FUNCTION_BLOCK FB_Dictionary IMPLEMENTS I_Dictionary
VAR_INPUT
END_VAR
VAR_OUTPUT
END_VAR
VAR
	bAdd:				BOOL;
	bReset:				Bool;
	bLoad:				BOOL;
	bSave:				BOOL;
	fbJson:				FB_JsonDomParser;
  	json:				SJsonValue;

	sJson: 				STRING(255);
END_VAR

IF bReset THEN
	bReset:= FALSE;
	json:= fbJson.NewDocument();
	bSave:= TRUE;
END_IF

IF bAdd THEN

	M_Add('member.Value1', 'Value');
	M_Add('member.Value2', 'Value');
	
END_IF


IF bLoad THEN
	fbJson.LoadDocumentFromFile('C:\Test.json', bLoad);
END_IF
IF bSave THEN
	fbJson.SaveDocumentToFile('C:\Test.json', bSave);
END_IF

fbJson.CopyDocument(sJson, SIZEOF(sJson));

METHOD PUBLIC M_Add : BOOL
VAR_INPUT
	Key:		STRING(255);
	Value:		STRING(255);
END_VAR
VAR 
	sKey:			String(255);
	nPosition:		INT;
END_VAR
//nPosition:= FIND(Key, '.')
//WHILE nPosition <> 0 DO
//	sKey:= LEFT(Key, nPosition);

//	nPosition:= FIND(Key, '.')
//END_WHILE

IF fbJson.FindMember(json, Key) = 0 THEN
	fbJson.AddStringMember(json, Key, Value);		
END_IF
END_METHOD

METHOD PUBLIC M_GetSTRING : String(255)
VAR_INPUT
	sName:	STRING(255);
END_VAR
END_METHOD

METHOD PUBLIC M_Load : BOOL
VAR_INPUT
	sFile:	STRING(255);
END_VAR
END_METHOD

METHOD PUBLIC M_Reset : BOOL
VAR_INPUT
END_VAR
END_METHOD

METHOD PUBLIC M_Save : BOOL
VAR_INPUT
END_VAR
END_METHOD

END_FUNCTION_BLOCK

(* stored: Version 1.1.0.1, ProductVersion 3.1.4024.12
   POU FB_Dictionary: Id {ca35913f-5cdc-0fb1-22b9-4c30741035cf}, SpecialFunc None
   Method M_Add: Id {5f198432-6b9a-0cc9-223e-32fac07c9c15}
   Method M_GetSTRING: Id {36d7e4d9-6385-0d15-1db3-61b9b3f66c18}
   Method M_Load: Id {0cfe07f9-80a6-0092-1199-05d47a634bea}
   Method M_Reset: Id {a41c1e35-f20d-09aa-09c0-ce2dae9cb17d}
   Method M_Save: Id {f15ba428-e316-0337-1810-7cf2e63511bb} *)
